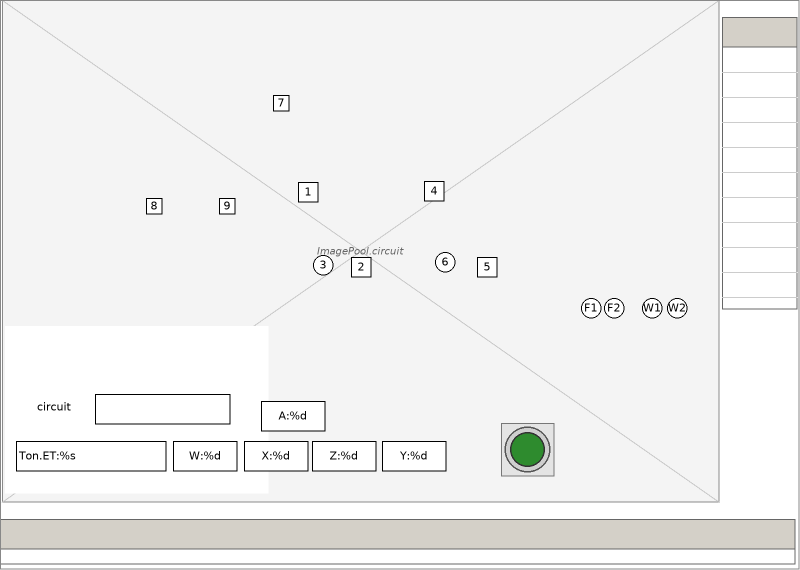
VISUALIZATION VIS_MU  // 800x570
    Image (2,0 717x502), image: ImagePool.circuit
    Ellipse (313,255 20x20), "3", colour toggle: stOutput.bqSubCircPumpWorking[1]
    Rectangle (351,257 20x20), "2", colour toggle: GVL.inklevel_W_L_BOT
        toggle stInput.biSubInkTankLevel[15]
    Ellipse (435,252 20x20), "6", colour toggle: stOutput.bqSubCircPumpWorking[2]
    Rectangle (477,257 20x20), "5", colour toggle: GVL.inklevel_W_R_BOT
        toggle stInput.biSubInkTankLevel[18]
    Rectangle (298,182 20x20), "1", colour toggle: GVL.inklevel_W_L_TOP
        toggle stInput.biSubInkTankLevel[16]
    Rectangle (424,181 20x20), "4", colour toggle: GVL.inklevel_W_R_TOP
        toggle stInput.biSubInkTankLevel[17]
    Rectangle (146,198 16x16), "8", colour toggle: stOutput.bqVacValve_W
    Rectangle (219,198 16x16), "9", colour toggle: stOutput.bqVacValve_C
    Rectangle (273,95 16x16), "7", colour toggle: stOutput.bqPurValve
    Ellipse (581,298 20x20), "F1", colour toggle: stOutput.bqFillPumpWorking[19]
    Ellipse (604,298 20x20), "F2", colour toggle: stOutput.bqFillPumpWorking[20]
    Ellipse (642,298 20x20), "W1", colour toggle: stOutput.bqFillPumpWorking[13]
    Ellipse (667,298 20x20), "W2", colour toggle: stOutput.bqFillPumpWorking[15]
    Rectangle (5,326 263x167)
    Table (0,519 795x45), data array: P_MaintenanceUnit.FB_Auto_Cycles_Swap
        p3854506369: P_MaintenanceUnit.FB_Auto_Cycles_Swap.Sensor1
        p1892666644: P_MaintenanceUnit.FB_Auto_Cycles_Swap.Sensor4
        p338671338: P_MaintenanceUnit.FB_Auto_Cycles_Swap.Circ_Pump_L
        p2170511999: P_MaintenanceUnit.FB_Auto_Cycles_Swap.Circ_Pump_R
        p3723444502: P_MaintenanceUnit.FB_Auto_Cycles_Swap.Circ_normal_error
        p1218418051: P_MaintenanceUnit.FB_Auto_Cycles_Swap.btPurge
        p746581629: P_MaintenanceUnit.FB_Auto_Cycles_Swap.state
        p3104783080: P_MaintenanceUnit.FB_Auto_Cycles_Swap.error_code
        p2501879983: P_MaintenanceUnit.FB_Auto_Cycles_Swap.SwapInfo
        p7306298: P_MaintenanceUnit.FB_Auto_Cycles_Swap.VacValve_V8
        p1933151965: P_MaintenanceUnit.FB_Auto_Cycles_Swap.PurValve_V7
        p3863566920: P_MaintenanceUnit.FB_Auto_Cycles_Swap.alternate_Pumping
        p2192122294: P_MaintenanceUnit.FB_Auto_Cycles_Swap.Swapping_Done
        p400160035: P_MaintenanceUnit.FB_Auto_Cycles_Swap.Error
        p1265227338: P_MaintenanceUnit.FB_Auto_Cycles_Swap.step
        p3726181087: P_MaintenanceUnit.FB_Auto_Cycles_Swap.stepA
        p3136911649: P_MaintenanceUnit.FB_Auto_Cycles_Swap.stepB1
        p797552052: P_MaintenanceUnit.FB_Auto_Cycles_Swap.stepB2
        p60375027: P_MaintenanceUnit.FB_Auto_Cycles_Swap.Ton
        p2531912550: P_MaintenanceUnit.FB_Auto_Cycles_Swap.ton7
        p693678525: P_MaintenanceUnit.FB_Auto_Cycles_Swap.ton10
        p3156763944: P_MaintenanceUnit.FB_Auto_Cycles_Swap.FB_SQUARE
        p3636993750: P_MaintenanceUnit.FB_Auto_Cycles_Swap.W
        p1303956035: P_MaintenanceUnit.FB_Auto_Cycles_Swap.X
        p285796650: P_MaintenanceUnit.FB_Auto_Cycles_Swap.A
        p2222472639: P_MaintenanceUnit.FB_Auto_Cycles_Swap.Z
        p3768075841: P_MaintenanceUnit.FB_Auto_Cycles_Swap.Y
        p1978176212: P_MaintenanceUnit.FB_Auto_Cycles_Swap.cycle_r_trig1
        p1509425299: P_MaintenanceUnit.FB_Auto_Cycles_Swap.cycle_r_trig2
        p3431519238: P_MaintenanceUnit.FB_Auto_Cycles_Swap.cycle_x1
        p2846402210: P_MaintenanceUnit.FB_Auto_Cycles_Swap.cycle_x2
        p1020817975: P_MaintenanceUnit.FB_Auto_Cycles_Swap.purge_F_trig
        p1480067529: P_MaintenanceUnit.FB_Auto_Cycles_Swap.dely_off_setoff
        p3444104540: P_MaintenanceUnit.FB_Auto_Cycles_Swap.dely_emstop
        p76032672: GVL_API.stMU.Initialize
        p1617449310: GVL_API.stMU.Swap
        p4112025035: P_MaintenanceUnit.FB_Auto_Cycles_Swap.CYCLE
        p3641186188: GVL_API.stMU.SetOff
        p633067465: initialize
        p1398730484: swap
        p3327948760: P_MaintenanceUnit.FB_Auto_Cycles_Swap.initialize
        p1777678866: P_MaintenanceUnit.FB_Auto_Cycles_Swap.swap
        p1879929205: P_MaintenanceUnit.FB_Auto_Cycles_Swap.setoff
        Columns.Column.[37].Template: OnMouseDown: write P_MaintenanceUnit.FB_Auto_Cycles_Swap.CYCLE via Default, min 0, max 1
        Columns.Column.[38].Template: toggle GVL_API.stMU.SetOff
        Columns.Column.[35].Template: toggle GVL_API.stMU.Initialize
        Columns.Column.[36].Template: toggle GVL_API.stMU.Swap
    Rectangle (16,441 150x30), "Ton.ET:%s", text variable: P_MaintenanceUnit.FB_Auto_Cycles_Swap.Ton.ET
    Table (722,17 75x292), data array: T
        p3854506369: T[INDEX]
        Columns.Column.[0].Template: OnMouseDown: write T[INDEX] via Default
    Rectangle (173,441 64x30), "W:%d", text variable: P_MaintenanceUnit.FB_Auto_Cycles_Swap.W
    Rectangle (244,441 64x30), "X:%d", text variable: P_MaintenanceUnit.FB_Auto_Cycles_Swap.X
    PushSwitch (500,423 55x53), variable: stInput.btPurge, behaviour: TAP, style: Switch-PushSwitch-Green
    Rectangle (312,441 64x30), "Z:%d", text variable: P_MaintenanceUnit.FB_Auto_Cycles_Swap.Z
    Rectangle (382,441 64x30), "Y:%d", text variable: P_MaintenanceUnit.FB_Auto_Cycles_Swap.Y
    Rectangle (95,394 135x30), text list: 'TextList_SubTank_circuit', text index: SubTankInk_type
        OnMouseDown: write HMI_CircPump1_V via Default, min 0, max 5
    Label (24,392 60x30), "circuit"
    Rectangle (261,401 64x30), "A:%d", text variable: P_MaintenanceUnit.FB_Auto_Cycles_Swap.A
END_VISUALIZATION

(* stored: Version 1.1.0.1, ProductVersion 3.1.4024.11
   Visu VIS_MU: Id {eec51cd6-ba0e-43c7-9b90-75dfcc9ec0d1} *)
